// TIA Portal V17 export
// export: Created 2025-06-26T06:49:12.7902383Z, ExportSetting WithDefaults, DisplayName Totally Integrated Automation Portal, DisplayVersion V17 Update 8, DisplayName TIA Portal Openness, DisplayVersion V17 Update 8, DisplayName TIA Portal Version Control Interface, DisplayVersion V17, DisplayName STEP 7 Professional, DisplayVersion V17 Update 8, DisplayName STEP 7 Safety, DisplayVersion V17 Update 6, DisplayName WinCC Advanced, DisplayVersion V17 Update 8
FUNCTION_BLOCK "ShaftSealCartridge"   // FB13, FBD
TITLE = Shaft seal cartridge
{ S7_Optimized_Access := 'TRUE' }
VERSION : 0.1
// stored: AutoNumber true, IsIECCheckEnabled false, IsRetainMemResEnabled false, MemoryReserve 100, SetENOAutomatically false, UDAEnableTagReadback false
   VAR_INPUT
      bEnable { ExternalAccessible := 'False'; ExternalVisible := 'False'; ExternalWritable := 'False'} : Bool;   // Enable from process. 1 = enabled, 0 = disabled.
      bReset { ExternalAccessible := 'False'; ExternalVisible := 'False'; ExternalWritable := 'False'} : Bool;
   END_VAR
   VAR
      Cooler { ExternalAccessible := 'False'; ExternalVisible := 'False'; ExternalWritable := 'False'} : "fbOnOffRegulator";
      Recharge { ExternalAccessible := 'False'; ExternalVisible := 'False'; ExternalWritable := 'False'; S7_SetPoint := 'True'} : "fbOnOffRegulator";
      A5257 { ExternalAccessible := 'False'; ExternalVisible := 'False'; ExternalWritable := 'False'; S7_SetPoint := 'True'} : "fbLowAlarm";
      A5258 { ExternalAccessible := 'False'; ExternalVisible := 'False'; ExternalWritable := 'False'; S7_SetPoint := 'True'} : "fbHighAlarm";
      A5259 { ExternalAccessible := 'False'; ExternalVisible := 'False'; ExternalWritable := 'False'; S7_SetPoint := 'True'} : "fbHighAlarm";
      A5260 { ExternalAccessible := 'False'; ExternalVisible := 'False'; ExternalWritable := 'False'; S7_SetPoint := 'True'} : "fbLowAlarm";
      A5261 { ExternalAccessible := 'False'; ExternalVisible := 'False'; ExternalWritable := 'False'; S7_SetPoint := 'True'} : "fbLowAlarm";
      A5262 { ExternalAccessible := 'False'; ExternalVisible := 'False'; ExternalWritable := 'False'; S7_SetPoint := 'True'} : "fbHighAlarm";
      A5263 { ExternalAccessible := 'False'; ExternalVisible := 'False'; ExternalWritable := 'False'; S7_SetPoint := 'True'} : "fbHighAlarm";
      A5268 { ExternalAccessible := 'False'; ExternalVisible := 'False'; ExternalWritable := 'False'; S7_SetPoint := 'True'} : "fbDigitalAlarm";
      nState { ExternalAccessible := 'False'; ExternalVisible := 'False'; ExternalWritable := 'False'; S7_SetPoint := 'True'} : USInt;
      bEnableAuto { ExternalAccessible := 'False'; ExternalVisible := 'False'; ExternalWritable := 'False'} : Bool;   // Circulation regulator is enabled in Auto
      bEnableCoolerAuto { ExternalAccessible := 'False'; ExternalVisible := 'False'; ExternalWritable := 'False'} : Bool;   // Cooling regulator is enabled in Auto
      bEnableRechargeAuto { ExternalAccessible := 'False'; ExternalVisible := 'False'; ExternalWritable := 'False'} : Bool;   // Recharging regulator is enabled in Auto
      bRunReqAuto { ExternalAccessible := 'False'; ExternalVisible := 'False'; ExternalWritable := 'False'} : Bool;   // Run in auto
      bStart { ExternalAccessible := 'False'; ExternalVisible := 'False'; ExternalWritable := 'False'} : R_TRIG;
   END_VAR
BEGIN

REGION Network 1: Delta-T over shaft seal
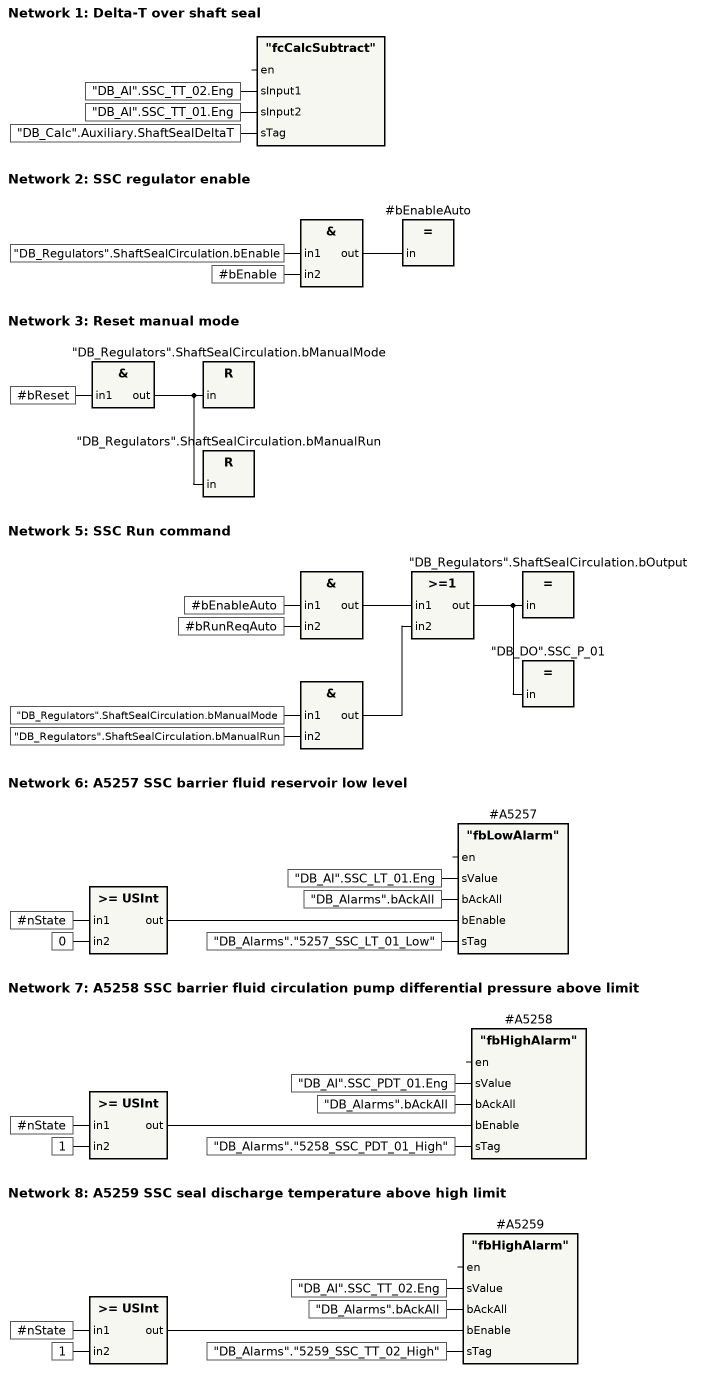
   "fcCalcSubtract"(sInput1 := "DB_AI".SSC_TT_02.Eng,
                    sInput2 := "DB_AI".SSC_TT_01.Eng,
                    sTag := "DB_Calc".Auxiliary.ShaftSealDeltaT);
END_REGION

REGION Network 2: SSC regulator enable
   // Start from input pin when enabled from HMI
   #bEnableAuto := "DB_Regulators".ShaftSealCirculation.bEnable AND #bEnable;
END_REGION

REGION Network 3: Reset manual mode
   IF #bReset THEN
       "DB_Regulators".ShaftSealCirculation.bManualMode := FALSE;
       "DB_Regulators".ShaftSealCirculation.bManualRun := FALSE;
   END_IF;
END_REGION

REGION Network 4 (SCL): SSC system state machine
   // Don't go into run state unless the pressure and temperature are first ok
   // Prevent retriggering
   #bStart(CLK := #bEnableAuto);

   CASE #nState OF

       0: // OFF
           #bEnableCoolerAuto := FALSE;
           #bEnableRechargeAuto := FALSE;
           #bRunReqAuto := FALSE;
           "DB_Regulators".ShaftSealCirculation.bFault := FALSE;
           IF #bStart.Q THEN
               #nState := 1;
           END_IF;
       1: // Startup. Wait for pressure and temperature to be ok
           #bEnableCoolerAuto := TRUE;
           #bEnableRechargeAuto := TRUE;
           //IF "DB_Regulators".ShaftSealCirculation.bEnable = FALSE THEN
           IF #bEnableAuto = FALSE THEN
               // Stop command
               #nState := 0;
           ELSIF "DB_Regulators".ShaftSealCirculation.bPressureLow AND "DB_Regulators".ShaftSealCirculation.bReservoirLow THEN
               // Barrier fluid pressure low and low fluid in recharge tank (can't recharge), give up.
               "DB_Regulators".ShaftSealCirculation.bFault := TRUE;
               #nState := 0;
           ELSIF "DB_Regulators".ShaftSealRecharge.bAtSetpoint AND "DB_Regulators".ShaftSealCooler.bAtSetpoint THEN
               // Pressure and temperature ok
               #nState := 2;
           END_IF;
       2: // Running
           #bRunReqAuto := TRUE;
           //IF "DB_Regulators".ShaftSealCirculation.bEnable = FALSE THEN
           IF #bEnableAuto = FALSE THEN
               // Stop command
               #nState := 0;
           END_IF;
           // Generate fault signal only in running state.
           "DB_Regulators".ShaftSealCirculation.bFault := "DB_Regulators".ShaftSealCirculation.bPressureLow OR "DB_Regulators".ShaftSealCirculation.bTemperatureHigh OR "DB_Regulators".ShaftSealCirculation.bDifferentialPressureHigh;
   END_CASE;
END_REGION

REGION Network 5: SSC Run command
   "DB_Regulators".ShaftSealCirculation.bOutput := (#bEnableAuto AND #bRunReqAuto) OR ("DB_Regulators".ShaftSealCirculation.bManualMode AND "DB_Regulators".ShaftSealCirculation.bManualRun);
   "DB_DO".SSC_P_01 := "DB_Regulators".ShaftSealCirculation.bOutput;
END_REGION

REGION Network 6: A5257 SSC barrier fluid reservoir low level
   // Always active
   #A5257(sValue := "DB_AI".SSC_LT_01.Eng,   // "fbLowAlarm"
          bAckAll := "DB_Alarms".bAckAll,
          bEnable := #nState >= 0,
          sTag := "DB_Alarms"."5257_SSC_LT_01_Low");
END_REGION

REGION Network 7: A5258 SSC barrier fluid circulation pump differential pressure above limit
   #A5258(sValue := "DB_AI".SSC_PDT_01.Eng,   // "fbHighAlarm"
          bAckAll := "DB_Alarms".bAckAll,
          bEnable := #nState >= 1,
          sTag := "DB_Alarms"."5258_SSC_PDT_01_High");
END_REGION

REGION Network 8: A5259 SSC seal discharge temperature above high limit
   #A5259(sValue := "DB_AI".SSC_TT_02.Eng,   // "fbHighAlarm"
          bAckAll := "DB_Alarms".bAckAll,
          bEnable := #nState >= 1,
          sTag := "DB_Alarms"."5259_SSC_TT_02_High");
END_REGION

REGION Network 9: A5260 SSC barrier fluid circulation pump suction temperature below low limit
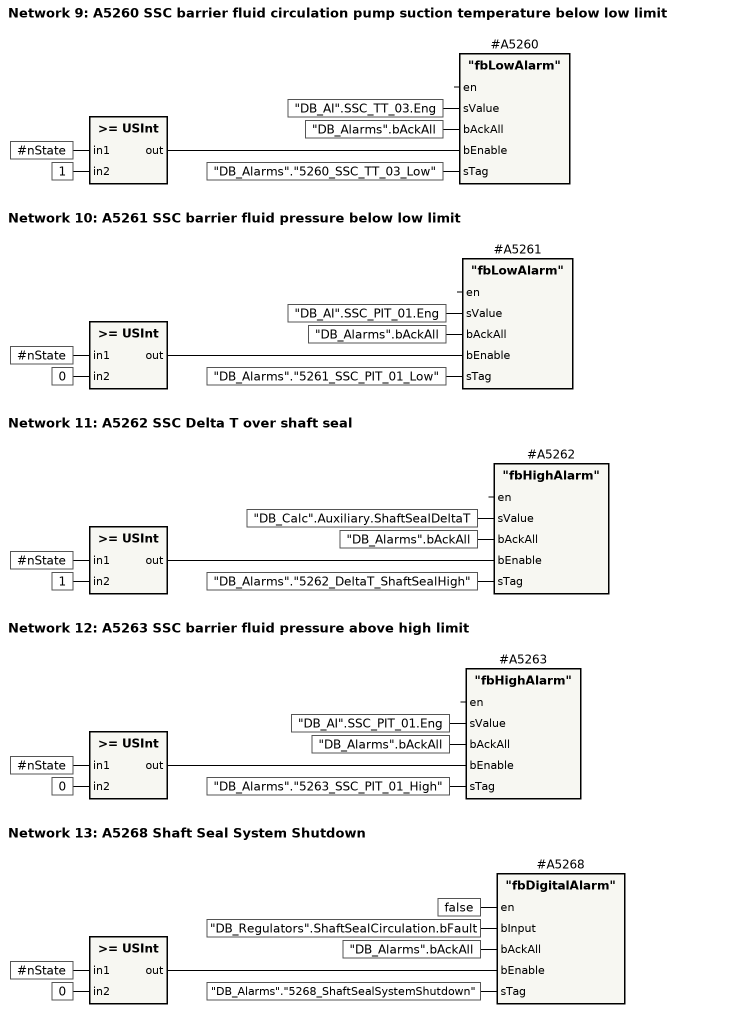
   #A5260(sValue := "DB_AI".SSC_TT_03.Eng,   // "fbLowAlarm"
          bAckAll := "DB_Alarms".bAckAll,
          bEnable := #nState >= 1,
          sTag := "DB_Alarms"."5260_SSC_TT_03_Low");
END_REGION

REGION Network 10: A5261 SSC barrier fluid pressure below low limit
   #A5261(sValue := "DB_AI".SSC_PIT_01.Eng,   // "fbLowAlarm"
          bAckAll := "DB_Alarms".bAckAll,
          bEnable := #nState >= 0,
          sTag := "DB_Alarms"."5261_SSC_PIT_01_Low");
END_REGION

REGION Network 11: A5262 SSC Delta T over shaft seal
   #A5262(sValue := "DB_Calc".Auxiliary.ShaftSealDeltaT,   // "fbHighAlarm"
          bAckAll := "DB_Alarms".bAckAll,
          bEnable := #nState >= 1,
          sTag := "DB_Alarms"."5262_DeltaT_ShaftSealHigh");
END_REGION

REGION Network 12: A5263 SSC barrier fluid pressure above high limit
   #A5263(sValue := "DB_AI".SSC_PIT_01.Eng,   // "fbHighAlarm"
          bAckAll := "DB_Alarms".bAckAll,
          bEnable := #nState >= 0,
          sTag := "DB_Alarms"."5263_SSC_PIT_01_High");
END_REGION

REGION Network 13: A5268 Shaft Seal System Shutdown
   // Regulator fault
   IF false THEN
       #A5268(bInput := "DB_Regulators".ShaftSealCirculation.bFault,   // "fbDigitalAlarm"
              bAckAll := "DB_Alarms".bAckAll,
              bEnable := #nState >= 0,
              sTag := "DB_Alarms"."5268_ShaftSealSystemShutdown");
   END_IF;
END_REGION

REGION Network 14: Faults
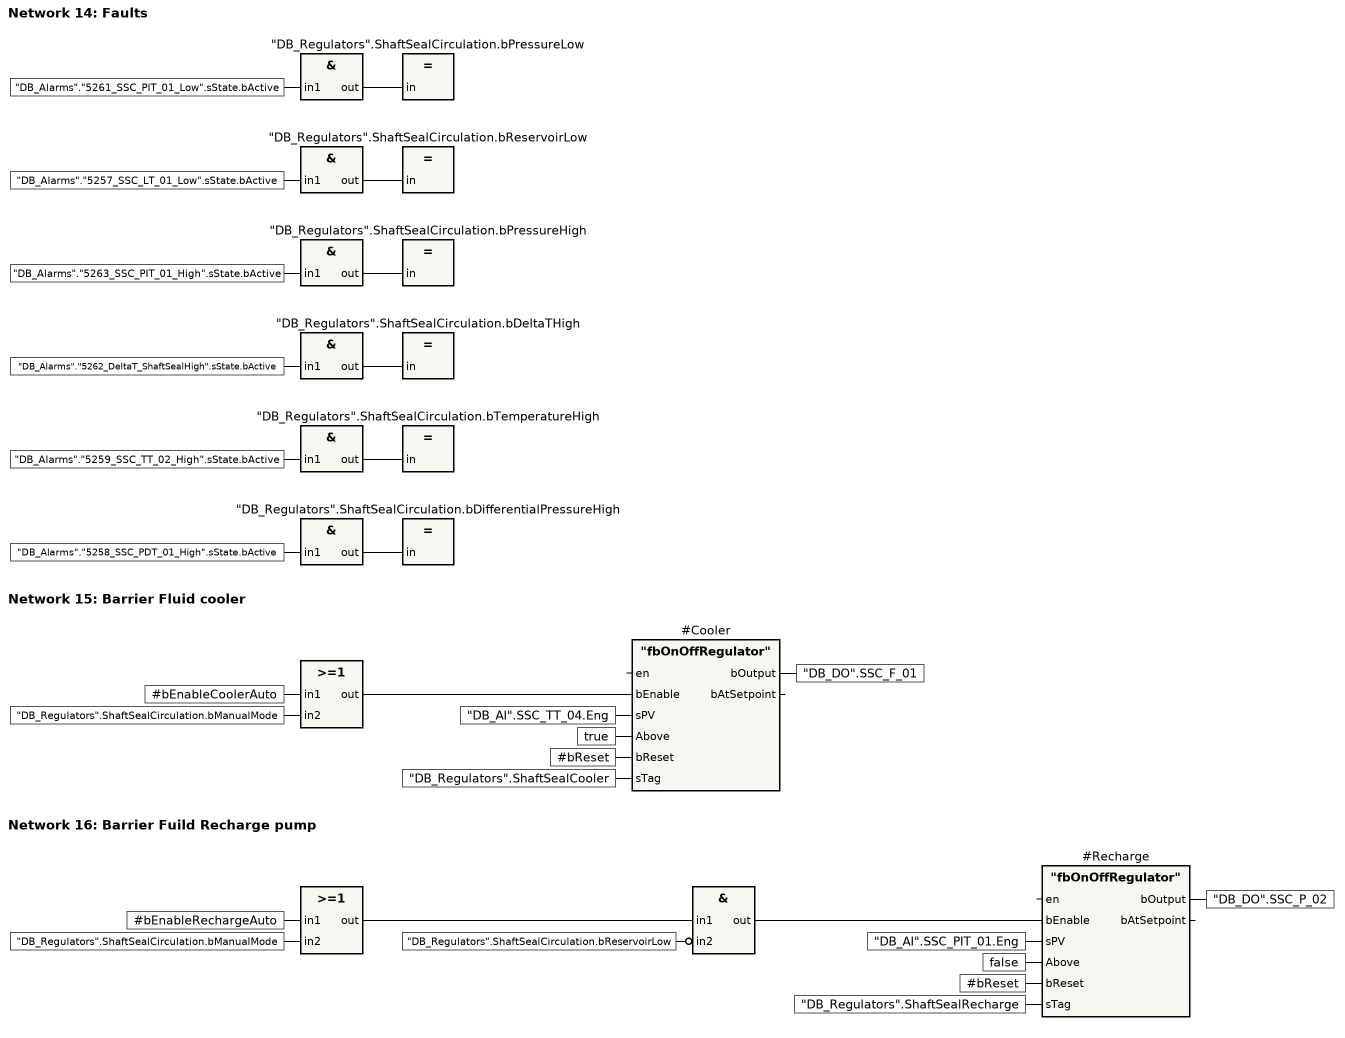
   "DB_Regulators".ShaftSealCirculation.bPressureLow := "DB_Alarms"."5261_SSC_PIT_01_Low".sState.bActive;
   "DB_Regulators".ShaftSealCirculation.bReservoirLow := "DB_Alarms"."5257_SSC_LT_01_Low".sState.bActive;
   "DB_Regulators".ShaftSealCirculation.bPressureHigh := "DB_Alarms"."5263_SSC_PIT_01_High".sState.bActive;
   "DB_Regulators".ShaftSealCirculation.bDeltaTHigh := "DB_Alarms"."5262_DeltaT_ShaftSealHigh".sState.bActive;
   "DB_Regulators".ShaftSealCirculation.bTemperatureHigh := "DB_Alarms"."5259_SSC_TT_02_High".sState.bActive;
   "DB_Regulators".ShaftSealCirculation.bDifferentialPressureHigh := "DB_Alarms"."5258_SSC_PDT_01_High".sState.bActive;
END_REGION

REGION Network 15: Barrier Fluid cooler
   // Run when the temperature in the barrier fluid gets too high
   #Cooler(bEnable := #bEnableCoolerAuto OR "DB_Regulators".ShaftSealCirculation.bManualMode,   // "fbOnOffRegulator"
           sPV := "DB_AI".SSC_TT_04.Eng,
           Above := true,
           bReset := #bReset,
           sTag := "DB_Regulators".ShaftSealCooler,
           bOutput => "DB_DO".SSC_F_01);
END_REGION

REGION Network 16: Barrier Fuild Recharge pump
   // Run when the pressure in the barrier fluid accumulator drops too low (and the reservoir is not empty)
   #Recharge(bEnable := (#bEnableRechargeAuto OR "DB_Regulators".ShaftSealCirculation.bManualMode) AND NOT "DB_Regulators".ShaftSealCirculation.bReservoirLow,   // "fbOnOffRegulator"
             sPV := "DB_AI".SSC_PIT_01.Eng,
             Above := false,
             bReset := #bReset,
             sTag := "DB_Regulators".ShaftSealRecharge,
             bOutput => "DB_DO".SSC_P_02);
END_REGION

REGION Network 17 (SCL)
   // Mode
   IF "DB_Regulators".ShaftSealCirculation.bManualMode = TRUE THEN
       "DB_Regulators".ShaftSealCirculation.nMode := 2;
   ELSIF "DB_Regulators".ShaftSealCirculation.bEnable = TRUE THEN
       "DB_Regulators".ShaftSealCirculation.nMode := 1;
   ELSE
       "DB_Regulators".ShaftSealCirculation.nMode := 0;
   END_IF;
END_REGION
END_FUNCTION_BLOCK
